Universal Robots URScript: Short_PHomeToInvB.script

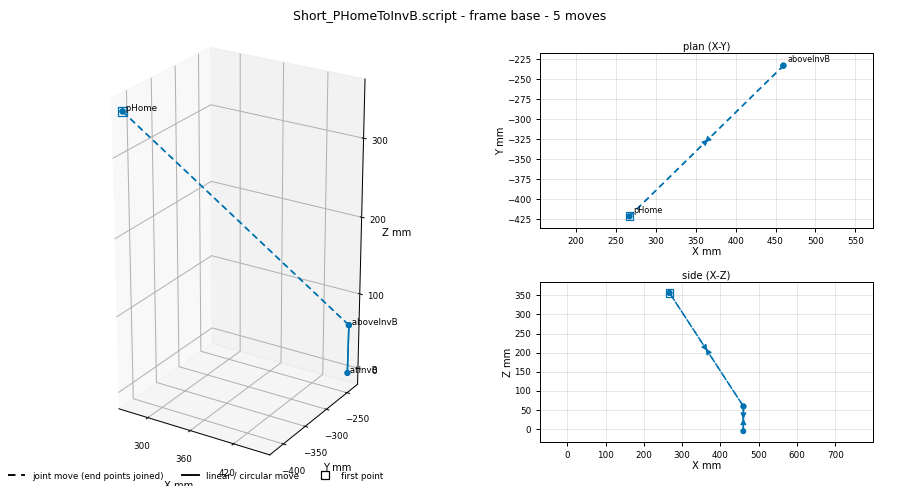
[picture p0: tool path of Short_PHomeToInvB.script in frame base, 5 of 5 moves have a stored position in this frame; points joined in program order, loops and branches not executed]
def Short_PHomeToInvB():
  set_gravity([0.0, 0.0, 9.82])
  set_tcp(p[0.0,0.0,0.076,0.7245313926163333,-1.7654607319513724,1.7638170400690123])
  set_payload(1.0)
  step_count_7255f790_e5c2_467f_85cd_3e9cf15fcca6 = 0.0
  thread Step_Counter_Thread_663b2e4f_e19b_465f_9f6b_c38d1401a853():
    while (True):
      step_count_7255f790_e5c2_467f_85cd_3e9cf15fcca6 = step_count_7255f790_e5c2_467f_85cd_3e9cf15fcca6 + 1.0
      sync()
    end
  end
  run Step_Counter_Thread_663b2e4f_e19b_465f_9f6b_c38d1401a853()
  set_standard_analog_input_domain(0, 0)
  set_standard_analog_input_domain(1, 0)
  set_tool_analog_input_domain(0, 1)
  set_tool_analog_input_domain(1, 1)
  set_analog_outputdomain(0, 0)
  set_analog_outputdomain(1, 0)
  set_input_actions_to_default()
  set_tool_voltage(0)
  modbus_add_signal("127.0.0.1", 255, 1, 3, "MODBUS_1", False)
  modbus_set_signal_update_frequency("MODBUS_1", 10)
  modbus_add_signal("127.0.0.1", 255, 203, 3, "MODBUS_2", False)
  modbus_set_signal_update_frequency("MODBUS_2", 10)
  modbus_set_runstate_dependent_choice("MODBUS_1",0)
  modbus_set_runstate_dependent_choice("MODBUS_2",0)
  set_safety_mode_transition_hardness(0)
  global stock_spacing=76.2
  global Gravity_Feeder=p[0.26545424739685874,-0.423573422243878,0.3571526050789449,0.1619581347920129,-0.4133494768613531,-2.317499916011395]
  global Linear_Slide=p[0.26542544581166166,-0.4235747955277341,0.35716918848305357,-0.010251867852105759,-0.0039919442596599315,-2.348075206071431]
  # begin: URCap Installation Node
  #   Source: VersaBuilt Robot2CNC, 2.0.9, VersaBuilt Robotics Inc.
  #   Type: R2C Config
  global vbSaveR2CIPAddr = "10.241.34.40"
  global vbSaveDoor = "SingleDoor"
  global vbSaveDoorSensors = True
  global vbSaveDoorWaitTime = 0
  global vbSaveViseSensors = True
  # end: URCap Installation Node
  def _adminLinearIndex2():
    $ 13 "_adminLinearIndex2" "noBreak"
    $ 14 "Move_linear_slide_Index2"
    $ 15 "var_1≔ False "
    global var_1=  False
    $ 16 "Loop var_1≟ False "
    while (var_1 ==   False  ):
      $ 17 "var_1≔socket_open('10.241.34.52',4001)"
      global var_1=socket_open("10.241.34.52",4001)
    end
    $ 18 "var_3≔1"
    global var_3=1
    $ 19 "Send≔'s r0x24 21'"
    global Send="s r0x24 21"
    $ 20 "socket_send_string(Send)"
    socket_send_string(Send)
    $ 21 "socket_send_byte(13)"
    socket_send_byte(13)
    $ 22 "Send_Reply≔socket_read_string()"
    global Send_Reply=socket_read_string()
    $ 23 "Send≔'s r0xca 56389'"
    global Send="s r0xca 56389"
    $ 24 "socket_send_string(Send)"
    socket_send_string(Send)
    $ 25 "socket_send_byte(13)"
    socket_send_byte(13)
    $ 26 "Send_Reply≔socket_read_string()"
    global Send_Reply=socket_read_string()
    $ 27 "Send≔'t 1'"
    global Send="t 1"
    $ 28 "socket_send_string(Send)"
    socket_send_string(Send)
    $ 29 "socket_send_byte(13)"
    socket_send_byte(13)
    $ 30 "Send_Reply≔socket_read_string()"
    global Send_Reply=socket_read_string()
    $ 31 "Loop var_3≠0"
    while (var_3 != 0):
      $ 32 "Send≔'g r0xA0'"
      global Send="g r0xA0"
      $ 33 "socket_send_string(Send)"
      socket_send_string(Send)
      $ 34 "socket_send_byte(13)"
      socket_send_byte(13)
      $ 35 "var_3≔socket_get_var('v')"
      global var_3=socket_get_var("v")
      $ 36 "Wait: 0.1"
      sleep(0.1)
    end
    $ 37 "socket_close()"
    socket_close()
    $ 38 "sync()"
    sync()
  end
  $ 1 "Robot Program"
  $ 2 "Call _adminLinearIndex2"
  _adminLinearIndex2()
  $ 3 "MoveJ"
  $ 4 "pHome" "breakAfter"
  movej(get_inverse_kin(p[.267143017205, -.421454805117, .355857452843, 1.113981300153, 1.106019241299, .005119613236], qnear=[-0.785346810017721, -1.570820156727926, -1.5707710425006312, -1.570820156727926, 1.5708600282669067, 1.3107746781315655E-4]), a=3.490658503988659, v=3.141592653589793)
  $ 5 "aboveInvB" "breakAfter"
  movej(get_inverse_kin(p[.460043718202, -.232619632006, .059707286805, 1.705964732826, -.008460135419, -1.211570608345], qnear=[-0.2543423811541956, -1.8824265638934534, -2.0373829046832483, -0.7959497610675257, 1.569312572479248, 2.1068875789642334]), a=3.490658503988659, v=3.141592653589793, r=0.048)
  $ 6 "MoveL"
  $ 7 "atInvB" "breakAfter"
  movel(p[.459620289343, -.233004510309, -.004986317020, 1.705964614413, -.008394298294, -1.211634670504], a=0.015, v=0.015)
  $ 8 "Set DO[0]=Off"
  set_standard_digital_out(0, False)
  $ 9 "Wait: 1.0"
  sleep(1.0)
  $ 10 "aboveInvB" "breakAfter"
  movel(p[.460043718202, -.232619632006, .059707286805, 1.705964732826, -.008460135419, -1.211570608345], a=0.015, v=0.015, r=0.05)
  $ 11 "MoveJ"
  $ 12 "pHome" "breakAfter"
  movej(get_inverse_kin(p[.267143017205, -.421454805117, .355857452843, 1.113981300153, 1.106019241299, .005119613236], qnear=[-0.785346810017721, -1.570820156727926, -1.5707710425006312, -1.570820156727926, 1.5708600282669067, 1.3107746781315655E-4]), a=1.7453292519943295, v=1.5707963267948966)
end
